FUNCTION_BLOCK EMA
VAR_INPUT
	NewValue: LREAL;
END_VAR
VAR_OUTPUT
	Value: LREAL;
END_VAR
VAR
	Weight: LREAL;
END_VAR

Value := Weight * NewValue + (1 - Weight) * Value;

METHOD FB_init : BOOL
VAR_INPUT
	bInitRetains : BOOL; // if TRUE, the retain variables are initialized (warm start / cold start)
	bInCopyCode : BOOL;  // if TRUE, the instance afterwards gets moved into the copy code (online change)
END_VAR
SetSampleCount(100);
END_METHOD

METHOD SetSampleCount : BOOL
VAR_INPUT
	n: int;
END_VAR
Weight := 2.0 / (1.0 + n);
END_METHOD

METHOD SetValue : BOOL
VAR_INPUT
	NewValue: LREAL;
END_VAR
Value := NewValue;
END_METHOD

END_FUNCTION_BLOCK

(* stored: Version 1.1.0.1, ProductVersion 3.1.4024.3
   POU EMA: Id {b98d6a3f-d2e9-4475-a7ba-2dd6a3a8821f}, SpecialFunc None
   Method FB_init: Id {4f362200-49e4-4aaa-b01f-f9b20fedbb24}
   Method SetSampleCount: Id {b4a3000f-dce9-4f1c-994a-db80cd1d7cd7}
   Method SetValue: Id {0b7f8250-5451-40ed-90e0-957159557063} *)
